TYPE U_APP_CTRL :
UNION
  stCtrl              : ST_APP_CTRL;
  byCtrl    AT %Q*    : ARRAY[1..SIZEOF(ST_APP_CTRL)] OF BYTE;
END_UNION
END_TYPE

(* stored: Version 1.1.0.1
   DUT U_APP_CTRL: Id {37071a30-676b-42f6-b5a0-376f15f85792} *)
